FUNCTION VERSION
  (* Standard: 61499-1; Description: Copyright (c) 2024 HR Agrartechnik GmbH This program and the accompanying materials are made available under the terms of the Eclipse Public License 2.0 which is available at https://www.eclipse.org/legal/epl-2.0/ SPDX-License-Identifier: EPL-2.0 *)
  (* Version 1.0, 2024-03-05, Franz Höpfinger, HR Agrartechnik GmbH *)
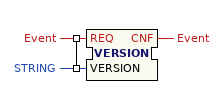
  EVENT_INPUT
    REQ WITH VERSION;
  END_EVENT
  EVENT_OUTPUT
    CNF;
  END_EVENT
  VAR_INPUT
    VERSION : STRING;
  END_VAR
  BODY IN ST:
FUNCTION VERSION
VAR_INPUT
	VERSION : STRING;
END_VAR
END_FUNCTION
  END_BODY
END_FUNCTION
